{attribute 'TcGenerated'}
// This function has been automatically generated from the project information.
VAR_GLOBAL CONSTANT
	{attribute 'const_non_replaced'}
	{attribute 'linkalways'}
	stLibVersion_Intecre_Utilities : ST_LibVersion := (iMajor := 1, iMinor := 7, iBuild := 0, iRevision := 0, sVersion := '1.7.0.0');
END_VAR

(* stored: Version 1.1.0.1, ProductVersion 3.1.4020.12
   GVL Global_Version: Id {868cbe4e-47d0-4354-9022-7dbbd9986b7d} *)
